// TIA Portal project "Assembler_Project" (V16)
// Vorlageprojekt für das Buch mit Zielsystem S7-1200

(* hardware
DEVICE "S7-1200-Station_1"  S7-1200 Station
   slot 0: "Baugruppenträger_0"  Rack  V1.0
   slot 1: "PLC_1"  CPU 1211C DC/DC/DC  6ES7 211-1AE40-0XB0  V4.1
*)

// ===== PLC "PLC_1"  CPU 1211C DC/DC/DC =====

VAR_GLOBAL   // PLC tag table "Standard-Variablentabelle"
   "Moving_X" AT %E0.0 : Bool;
   "Moving_Z" AT %E0.1 : Bool;
   "Start" AT %I1.2 : Bool;
   "Stop" AT %I1.4 : Bool;
   "Auto" AT %I1.6 : Bool;
   "Start_light" AT %Q1.1 : Bool;
   "Move_X" AT %Q0.0 : Bool;
   "Move_Z" AT %Q0.1 : Bool;
   "Grab" AT %Q0.2 : Bool;
   "Lid_conveyor" AT %Q0.3 : Bool;
   "Clamp lid" AT %Q0.4 : Bool;
   "Raise_lid_block" AT %Q0.5 : Bool;
   "Base_conveyor" AT %Q0.6 : Bool;
   "Clamp_base" AT %Q0.7 : Bool;
   "Raise_base_block" AT %Q1.0 : Bool;
   "Reset_light" AT %Q1.2 : Bool;
   "Stop_light" AT %Q1.3 : Bool;
   "Lid_block_raised" AT %I0.5 : Bool;
   "Set_System_State" AT %Q2.0 : Bool;
   "Item_detected" AT %I0.2 : Bool;
   "Lid_at_place" AT %I0.3 : Bool;
   "Lid_clamped" AT %I0.4 : Bool;
   "Base_at_place" AT %I0.6 : Bool;
   "Base_clamped" AT %I0.7 : Bool;
   "Base_block_raised" AT %I1.0 : Bool;
   "Assembled_parts_leaving" AT %I1.1 : Bool;
   "Emergency_stop" AT %I1.5 : Bool;
   "System_State" AT %M0.0 : Bool;
   "Lid_at_place_memory" AT %M0.1 : Bool;
   "Base_at_place_memory" AT %M0.2 : Bool;
   "Base_part_to_be_clamped" AT %M0.3 : Bool;
   "Lid_part_to_be_clamped" AT %M0.4 : Bool;
   "Reset" AT %I1.3 : Bool;
   "Moving_X_memory" AT %M0.6 : Bool;
   "Moving_-Z_memory1" AT %M0.7 : Bool;
   "Lid_part_grasped" AT %M1.7 : Bool;
   "Assembling_parts" AT %M0.5 : Bool;
   "Lid_part_lifted" AT %M2.0 : Bool;
   "Lid_part_moved_in_XDirection" AT %M2.1 : Bool;
   "Lid_part_lowered" AT %M2.2 : Bool;
   "Lid_part_dropped" AT %M2.3 : Bool;
   "Reset_assembly_memories" AT %M1.5 : Bool;
   "Assembled_parts_leaving_memory" AT %M1.4 : Bool;
   "Base_block_raised_memory" AT %M1.3 : Bool;
   "Lift_arm_after_assemble" AT %M2.4 : Bool;
   "Arm_dropped_to_grasp_lid" AT %M1.6 : Bool;
   "Moving_+Z_memory1" AT %M1.1 : Bool;
   "Moving_-Z_memory2" AT %M1.0 : Bool;
   "Moving_+Z_memory2" AT %M1.2 : Bool;
END_VAR

FUNCTION "Assemble" : Void   // FC2, LAD
{ S7_Optimized_Access := 'TRUE' }
VERSION : 0.1
   VAR_TEMP   // added for the SCL form of the ladder/FBD networks
      _w1 : Bool;
   END_VAR
BEGIN

REGION Network 1
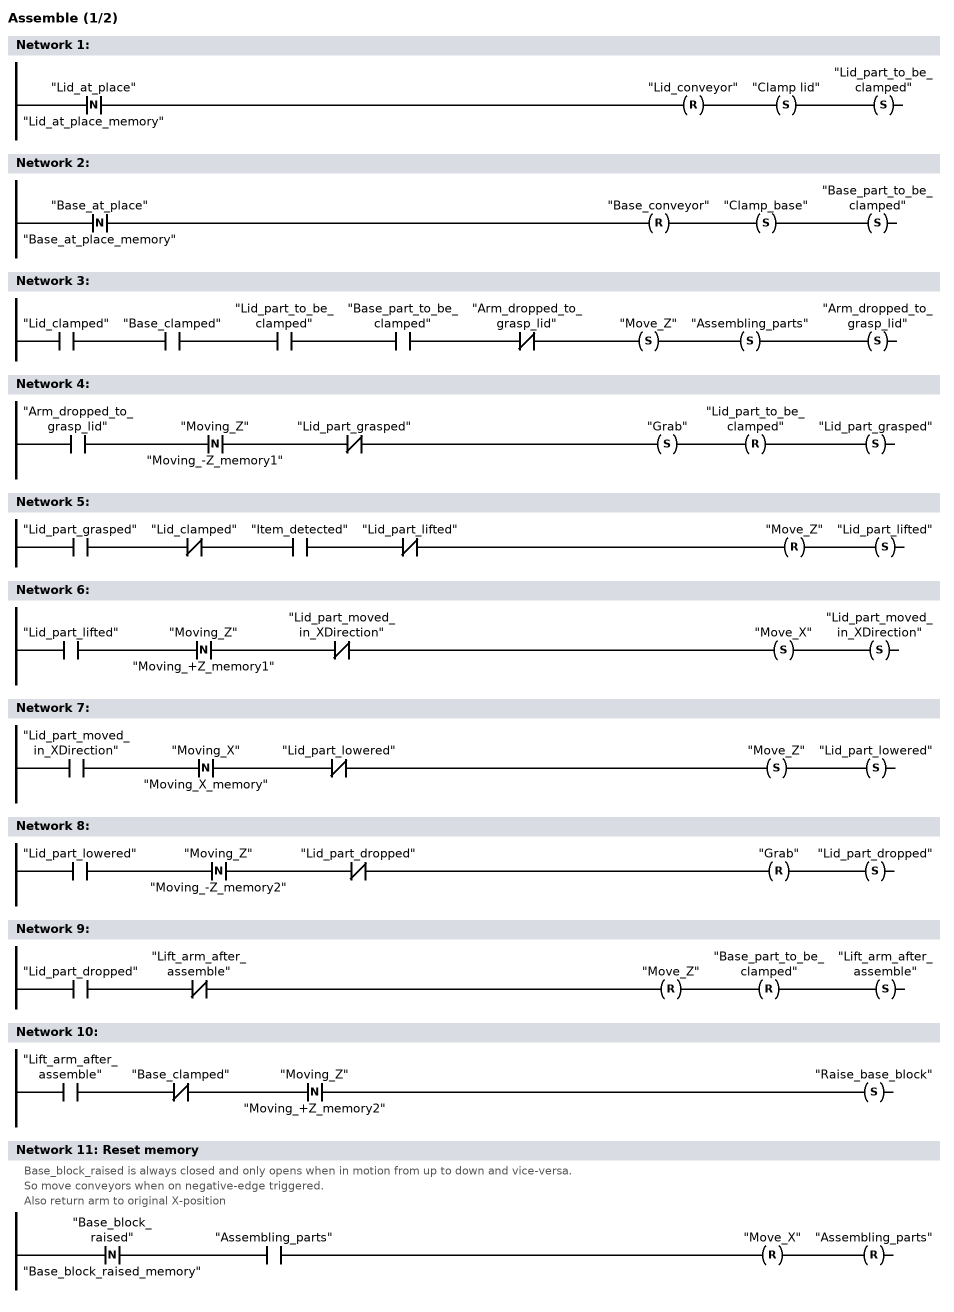
   RUNG wire#powerrail
      N_Contact(operand := "Lid_at_place", bit := "Lid_at_place_memory")
      R_Coil( "Lid_conveyor" )
      S_Coil( "Clamp lid" )
      S_Coil( "Lid_part_to_be_clamped" )
   END_RUNG
   // the same network as SCL:
   #_w1 := NOT "Lid_at_place" AND "Lid_at_place_memory";   // falling edge of "Lid_at_place"
   "Lid_at_place_memory" := "Lid_at_place";
   IF #_w1 THEN
       "Lid_conveyor" := FALSE;
       "Clamp lid" := TRUE;
       "Lid_part_to_be_clamped" := TRUE;
   END_IF;
END_REGION

REGION Network 2
   RUNG wire#powerrail
      N_Contact(operand := "Base_at_place", bit := "Base_at_place_memory")
      R_Coil( "Base_conveyor" )
      S_Coil( "Clamp_base" )
      S_Coil( "Base_part_to_be_clamped" )
   END_RUNG
   // the same network as SCL:
   #_w1 := NOT "Base_at_place" AND "Base_at_place_memory";   // falling edge of "Base_at_place"
   "Base_at_place_memory" := "Base_at_place";
   IF #_w1 THEN
       "Base_conveyor" := FALSE;
       "Clamp_base" := TRUE;
       "Base_part_to_be_clamped" := TRUE;
   END_IF;
END_REGION

REGION Network 3
   RUNG wire#powerrail
      Contact( "Lid_clamped" )
      Contact( "Base_clamped" )
      Contact( "Lid_part_to_be_clamped" )
      Contact( "Base_part_to_be_clamped" )
      I_Contact( "Arm_dropped_to_grasp_lid" )
      S_Coil( "Move_Z" )
      S_Coil( "Assembling_parts" )
      S_Coil( "Arm_dropped_to_grasp_lid" )
   END_RUNG
   // the same network as SCL:
   IF "Lid_clamped" AND "Base_clamped" AND "Lid_part_to_be_clamped" AND "Base_part_to_be_clamped" AND NOT "Arm_dropped_to_grasp_lid" THEN
       "Move_Z" := TRUE;
       "Assembling_parts" := TRUE;
       "Arm_dropped_to_grasp_lid" := TRUE;
   END_IF;
END_REGION

REGION Network 4
   RUNG wire#powerrail
      Contact( "Arm_dropped_to_grasp_lid" )
      N_Contact(operand := "Moving_Z", bit := "Moving_-Z_memory1")
      I_Contact( "Lid_part_grasped" )
      S_Coil( "Grab" )
      R_Coil( "Lid_part_to_be_clamped" )
      S_Coil( "Lid_part_grasped" )
   END_RUNG
   // the same network as SCL:
   #_w1 := "Arm_dropped_to_grasp_lid" AND NOT "Moving_Z" AND "Moving_-Z_memory1";   // falling edge of "Moving_Z"
   "Moving_-Z_memory1" := "Moving_Z";
   IF #_w1 AND NOT "Lid_part_grasped" THEN
       "Grab" := TRUE;
       "Lid_part_to_be_clamped" := FALSE;
       "Lid_part_grasped" := TRUE;
   END_IF;
END_REGION

REGION Network 5
   RUNG wire#powerrail
      Contact( "Lid_part_grasped" )
      I_Contact( "Lid_clamped" )
      Contact( "Item_detected" )
      I_Contact( "Lid_part_lifted" )
      R_Coil( "Move_Z" )
      S_Coil( "Lid_part_lifted" )
   END_RUNG
   // the same network as SCL:
   IF "Lid_part_grasped" AND NOT "Lid_clamped" AND "Item_detected" AND NOT "Lid_part_lifted" THEN
       "Move_Z" := FALSE;
       "Lid_part_lifted" := TRUE;
   END_IF;
END_REGION

REGION Network 6
   RUNG wire#powerrail
      Contact( "Lid_part_lifted" )
      N_Contact(operand := "Moving_Z", bit := "Moving_+Z_memory1")
      I_Contact( "Lid_part_moved_in_XDirection" )
      S_Coil( "Move_X" )
      S_Coil( "Lid_part_moved_in_XDirection" )
   END_RUNG
   // the same network as SCL:
   #_w1 := "Lid_part_lifted" AND NOT "Moving_Z" AND "Moving_+Z_memory1";   // falling edge of "Moving_Z"
   "Moving_+Z_memory1" := "Moving_Z";
   IF #_w1 AND NOT "Lid_part_moved_in_XDirection" THEN
       "Move_X" := TRUE;
       "Lid_part_moved_in_XDirection" := TRUE;
   END_IF;
END_REGION

REGION Network 7
   RUNG wire#powerrail
      Contact( "Lid_part_moved_in_XDirection" )
      N_Contact(operand := "Moving_X", bit := "Moving_X_memory")
      I_Contact( "Lid_part_lowered" )
      S_Coil( "Move_Z" )
      S_Coil( "Lid_part_lowered" )
   END_RUNG
   // the same network as SCL:
   #_w1 := "Lid_part_moved_in_XDirection" AND NOT "Moving_X" AND "Moving_X_memory";   // falling edge of "Moving_X"
   "Moving_X_memory" := "Moving_X";
   IF #_w1 AND NOT "Lid_part_lowered" THEN
       "Move_Z" := TRUE;
       "Lid_part_lowered" := TRUE;
   END_IF;
END_REGION

REGION Network 8
   RUNG wire#powerrail
      Contact( "Lid_part_lowered" )
      N_Contact(operand := "Moving_Z", bit := "Moving_-Z_memory2")
      I_Contact( "Lid_part_dropped" )
      R_Coil( "Grab" )
      S_Coil( "Lid_part_dropped" )
   END_RUNG
   // the same network as SCL:
   #_w1 := "Lid_part_lowered" AND NOT "Moving_Z" AND "Moving_-Z_memory2";   // falling edge of "Moving_Z"
   "Moving_-Z_memory2" := "Moving_Z";
   IF #_w1 AND NOT "Lid_part_dropped" THEN
       "Grab" := FALSE;
       "Lid_part_dropped" := TRUE;
   END_IF;
END_REGION

REGION Network 9
   RUNG wire#powerrail
      Contact( "Lid_part_dropped" )
      I_Contact( "Lift_arm_after_assemble" )
      R_Coil( "Move_Z" )
      R_Coil( "Base_part_to_be_clamped" )
      S_Coil( "Lift_arm_after_assemble" )
   END_RUNG
   // the same network as SCL:
   IF "Lid_part_dropped" AND NOT "Lift_arm_after_assemble" THEN
       "Move_Z" := FALSE;
       "Base_part_to_be_clamped" := FALSE;
       "Lift_arm_after_assemble" := TRUE;
   END_IF;
END_REGION

REGION Network 10
   RUNG wire#powerrail
      Contact( "Lift_arm_after_assemble" )
      I_Contact( "Base_clamped" )
      N_Contact(operand := "Moving_Z", bit := "Moving_+Z_memory2")
      S_Coil( "Raise_base_block" )
   END_RUNG
   // the same network as SCL:
   #_w1 := "Lift_arm_after_assemble" AND NOT "Base_clamped" AND NOT "Moving_Z" AND "Moving_+Z_memory2";   // falling edge of "Moving_Z"
   "Moving_+Z_memory2" := "Moving_Z";
   IF #_w1 THEN "Raise_base_block" := TRUE; END_IF;
END_REGION

REGION Network 11: Reset memory
   // Base_block_raised is always closed and only opens when in motion from up to down and vice-versa.
   // So move conveyors when on negative-edge triggered. 
   // Also return arm to original X-position
   RUNG wire#powerrail
      N_Contact(operand := "Base_block_raised", bit := "Base_block_raised_memory")
      Contact( "Assembling_parts" )
      R_Coil( "Move_X" )
      R_Coil( "Assembling_parts" )
   END_RUNG
   // the same network as SCL:
   #_w1 := NOT "Base_block_raised" AND "Base_block_raised_memory";   // falling edge of "Base_block_raised"
   "Base_block_raised_memory" := "Base_block_raised";
   IF #_w1 AND "Assembling_parts" THEN
       "Move_X" := FALSE;
       "Assembling_parts" := FALSE;
   END_IF;
END_REGION

REGION Network 12
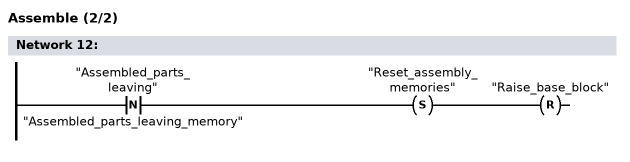
   RUNG wire#powerrail
      N_Contact(operand := "Assembled_parts_leaving", bit := "Assembled_parts_leaving_memory")
      S_Coil( "Reset_assembly_memories" )
      R_Coil( "Raise_base_block" )
   END_RUNG
   // the same network as SCL:
   #_w1 := NOT "Assembled_parts_leaving" AND "Assembled_parts_leaving_memory";   // falling edge of "Assembled_parts_leaving"
   "Assembled_parts_leaving_memory" := "Assembled_parts_leaving";
   IF #_w1 THEN
       "Reset_assembly_memories" := TRUE;
       "Raise_base_block" := FALSE;
   END_IF;
END_REGION
END_FUNCTION

FUNCTION "MHJ-PLC-Lab-Function-S71200" : Void   // FC9000, SCL
{ S7_Optimized_Access := 'TRUE' }
VERSION : 0.1
   VAR_TEMP
      rdTimeReturn : Int;
      outputTime : DTL;
      SyncVal : Byte;
      forVal : Int;
      forVal_2 : Int;
      Value : Byte;
   END_VAR
   VAR CONSTANT
      CompVal : Byte := 16#34;
      Value_01 : Byte := 16#11;
      Value_01_DW : DWord := 16#A165_D992;
      Value_02_DW : DWord := 16#58BE_4401;
   END_VAR
BEGIN

   #Value:=PEEK(area := 16#82,
        dbNumber := 0,
        byteOffset := 511);
   #Value := #Value + 1;

   POKE(area := 16#82,
        dbNumber := 0,
        byteOffset := 511,
        value := #Value);

   POKE(area:=16#81,
        dbNumber:=0,
        byteOffset:=1016,
        value:=#Value_01_DW);
   POKE(area := 16#81,
        dbNumber := 0,
        byteOffset := 1020,
        value := #Value_02_DW);

   POKE(area := 16#81,
        dbNumber := 0,
        byteOffset := 511,
        value := B#16#00);

   FOR #forVal := 0 TO 120 DO
       FOR #forVal_2:=0 TO 10 DO
           #rdTimeReturn:=RD_SYS_T(#outputTime);
           #rdTimeReturn := WR_SYS_T(#outputTime);
           #rdTimeReturn := RD_SYS_T(#outputTime);
           #rdTimeReturn := WR_SYS_T(#outputTime);
       END_FOR;
       #SyncVal:= PEEK(area := 16#81,
                      dbNumber := 0,
                      byteOffset := 511);
       IF #SyncVal = #CompVal THEN
          GOTO M_1;
       END_IF;
   END_FOR;
   RETURN;

   M_1:
   POKE(area := 16#81,
        dbNumber := 0,
        byteOffset := 511,
        value := B#16#0);
END_FUNCTION

ORGANIZATION_BLOCK "Main"   // OB1, LAD, ProgramCycle
TITLE = "Main Program Sweep (Cycle)"
{ S7_Optimized_Access := 'TRUE' }
VERSION : 0.1
   VAR_INPUT
      Initial_Call : Bool;   // Initial call of this OB
      Remanence : Bool;   // =True, if remanent data are available
   END_VAR
BEGIN

REGION Network 1: Konnektierungsbaustein für PLC-Lab
   // Im Netzwerk 1 wird der Konnektierungsbaustein für PLC-Lab aufgerufen.
   // Dieser Aufruf darf nicht entfernt werden!
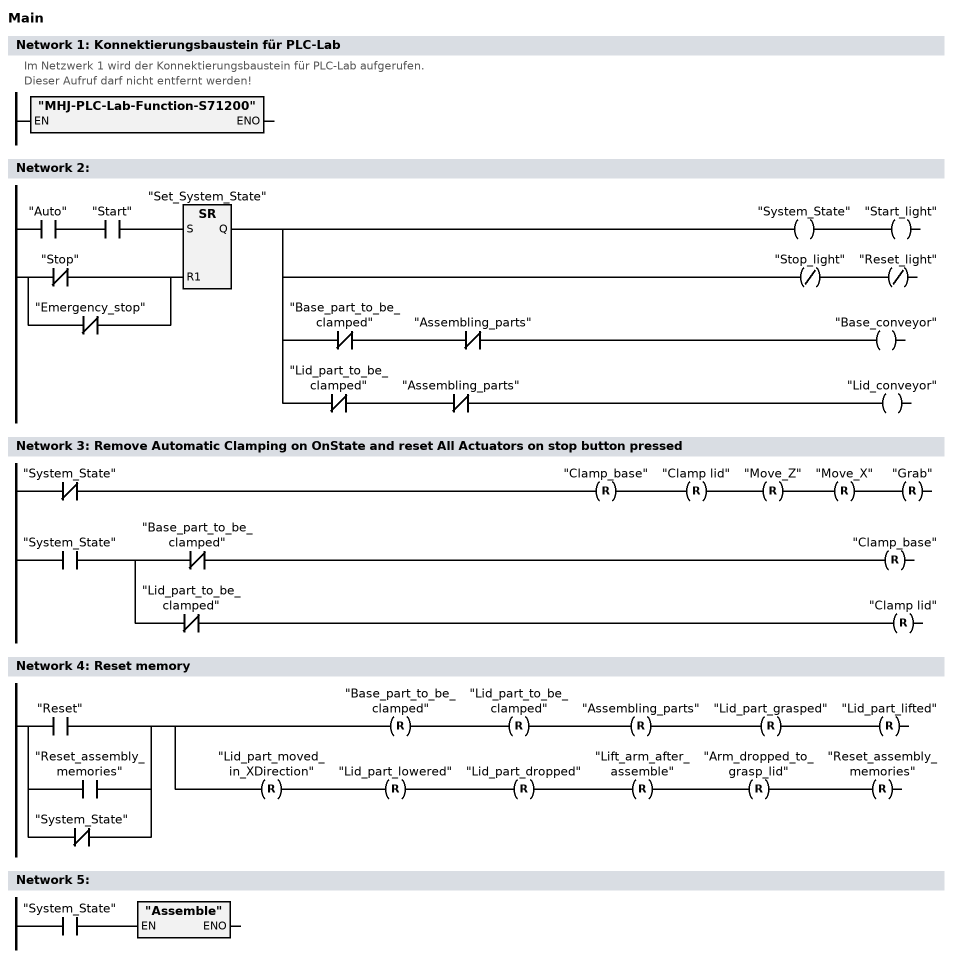
   RUNG wire#powerrail
      "MHJ-PLC-Lab-Function-S71200"()
   END_RUNG
   // the same network as SCL:
   "MHJ-PLC-Lab-Function-S71200"();
END_REGION

REGION Network 2
   RUNG wire#powerrail
      Contact( "Auto" )
      Contact( "Start" )
      S_SR(operand := "Set_System_State", r1 := wire#w1)
      wire#w2
      Coil( "System_State" )
      Coil( "Start_light" )
   END_RUNG
   RUNG wire#powerrail
      I_Contact( "Stop" )
   END_RUNG wire#w1
   RUNG wire#powerrail
      I_Contact( "Emergency_stop" )
   END_RUNG wire#w1
   RUNG wire#w2
      I_Coil( "Stop_light" )
      I_Coil( "Reset_light" )
   END_RUNG
   RUNG wire#w2
      I_Contact( "Base_part_to_be_clamped" )
      I_Contact( "Assembling_parts" )
      Coil( "Base_conveyor" )
   END_RUNG
   RUNG wire#w2
      I_Contact( "Lid_part_to_be_clamped" )
      I_Contact( "Assembling_parts" )
      Coil( "Lid_conveyor" )
   END_RUNG
   // the same network as SCL:
   IF "Auto" AND "Start" THEN
       "Set_System_State" := TRUE;   // SR flip-flop
   END_IF;
   IF NOT "Stop" OR NOT "Emergency_stop" THEN "Set_System_State" := FALSE; END_IF;
   "System_State" := "Set_System_State";
   "Start_light" := "Set_System_State";
   "Stop_light" := NOT "Set_System_State";
   "Reset_light" := NOT "Set_System_State";
   "Base_conveyor" := "Set_System_State" AND NOT "Base_part_to_be_clamped" AND NOT "Assembling_parts";
   "Lid_conveyor" := "Set_System_State" AND NOT "Lid_part_to_be_clamped" AND NOT "Assembling_parts";
END_REGION

REGION Network 3: Remove Automatic Clamping on OnState and reset All Actuators on stop button pressed
   RUNG wire#powerrail
      I_Contact( "System_State" )
      R_Coil( "Clamp_base" )
      R_Coil( "Clamp lid" )
      R_Coil( "Move_Z" )
      R_Coil( "Move_X" )
      R_Coil( "Grab" )
   END_RUNG
   RUNG wire#powerrail
      Contact( "System_State" )
      wire#w1
      I_Contact( "Base_part_to_be_clamped" )
      R_Coil( "Clamp_base" )
   END_RUNG
   RUNG wire#w1
      I_Contact( "Lid_part_to_be_clamped" )
      R_Coil( "Clamp lid" )
   END_RUNG
   // the same network as SCL:
   IF NOT "System_State" THEN
       "Clamp_base" := FALSE;
       "Clamp lid" := FALSE;
       "Move_Z" := FALSE;
       "Move_X" := FALSE;
       "Grab" := FALSE;
   END_IF;
   IF "System_State" AND NOT "Base_part_to_be_clamped" THEN "Clamp_base" := FALSE; END_IF;
   IF "System_State" AND NOT "Lid_part_to_be_clamped" THEN "Clamp lid" := FALSE; END_IF;
END_REGION

REGION Network 4: Reset memory
   RUNG wire#powerrail
      Contact( "Reset" )
      wire#w1
      R_Coil( "Base_part_to_be_clamped" )
      R_Coil( "Lid_part_to_be_clamped" )
      R_Coil( "Assembling_parts" )
      R_Coil( "Lid_part_grasped" )
      R_Coil( "Lid_part_lifted" )
   END_RUNG
   RUNG wire#powerrail
      Contact( "Reset_assembly_memories" )
   END_RUNG wire#w1
   RUNG wire#powerrail
      I_Contact( "System_State" )
   END_RUNG wire#w1
   RUNG wire#w1
      R_Coil( "Lid_part_moved_in_XDirection" )
      R_Coil( "Lid_part_lowered" )
      R_Coil( "Lid_part_dropped" )
      R_Coil( "Lift_arm_after_assemble" )
      R_Coil( "Arm_dropped_to_grasp_lid" )
      R_Coil( "Reset_assembly_memories" )
   END_RUNG
   // the same network as SCL:
   IF "Reset" OR "Reset_assembly_memories" OR NOT "System_State" THEN
       "Base_part_to_be_clamped" := FALSE;
       "Lid_part_to_be_clamped" := FALSE;
       "Assembling_parts" := FALSE;
       "Lid_part_grasped" := FALSE;
       "Lid_part_lifted" := FALSE;
       "Lid_part_moved_in_XDirection" := FALSE;
       "Lid_part_lowered" := FALSE;
       "Lid_part_dropped" := FALSE;
       "Lift_arm_after_assemble" := FALSE;
       "Arm_dropped_to_grasp_lid" := FALSE;
       "Reset_assembly_memories" := FALSE;
   END_IF;
END_REGION

REGION Network 5
   RUNG wire#powerrail
      Contact( "System_State" )
      "Assemble"()
   END_RUNG
   // the same network as SCL:
   IF "System_State" THEN "Assemble"(); END_IF;
END_REGION
END_ORGANIZATION_BLOCK